(* PLC project Unnamed, Unknown Unnamed 1 *)
(* stored: creationDateTime 2026-06-06T03:01:27, modificationDateTime 2026-06-06T03:01:27 *)

PROGRAM main
  VAR
    conveyor AT %QX0.0 : BOOL;  (* the entry conveyor that transport the boxes to the chain transfer *)
    Load AT %QX0.1 : BOOL;  (* the conveyor on the chain transfer that move the boxes to the right place to be then transported *)
    TransferLeft AT %QX0.3 : BOOL;  (* moves the boxes on the chain transfer to the left *)
    TransferRight AT %QX0.4 : BOOL;  (* moves the boxes on the chain transfer to the right *)
    ConveyoerLeft AT %QX0.5 : BOOL;  (* moves the short boxes to the remover where they get disposed *)
    conveyorRight AT %QX0.6 : BOOL;  (* moves the tall boxes to the remover where they get disposed *)
    HighSensor AT %IX0.0 : BOOL;  (* detects if the boxes are tall *)
    LowSensor AT %IX0.1 : BOOL;  (* detects if the boxes are tall ( the high sensor also need to be false for this to be useful ) *)
    PalletSensor AT %IX0.2 : BOOL;  (* detects the pallet to know to when to start the transportation *)
    Loaded AT %IX0.3 : BOOL;  (* sensor to detect the box is in the right place to be transported *)
    LeftEntry AT %IX0.4 : BOOL;  (* A sensor to to detect that the box has left the chain transfer and reached the left conveyor *)
    at_right_entry AT %IX0.6 : BOOL;  (* A sensor to to detect that the box has left the chain transfer and reached the right conveyor *)
  END_VAR
  VAR
    highsensor_memorybit : BOOL;  (* a boolean variable to save the state of the tall boxes *)
    lowsensor_memorybit : BOOL;  (* a boolean variable to save the state of the short boxes *)
    F_TRIG0 : F_TRIG;
    F_TRIG1 : F_TRIG;
    F_TRIG2 : F_TRIG;
    F_TRIG3 : F_TRIG;
    F_TRIG4 : F_TRIG;
    F_TRIG5 : F_TRIG;
    F_TRIG6 : F_TRIG;
    F_TRIG7 : F_TRIG;
    R_TRIG0 : R_TRIG;
  END_VAR

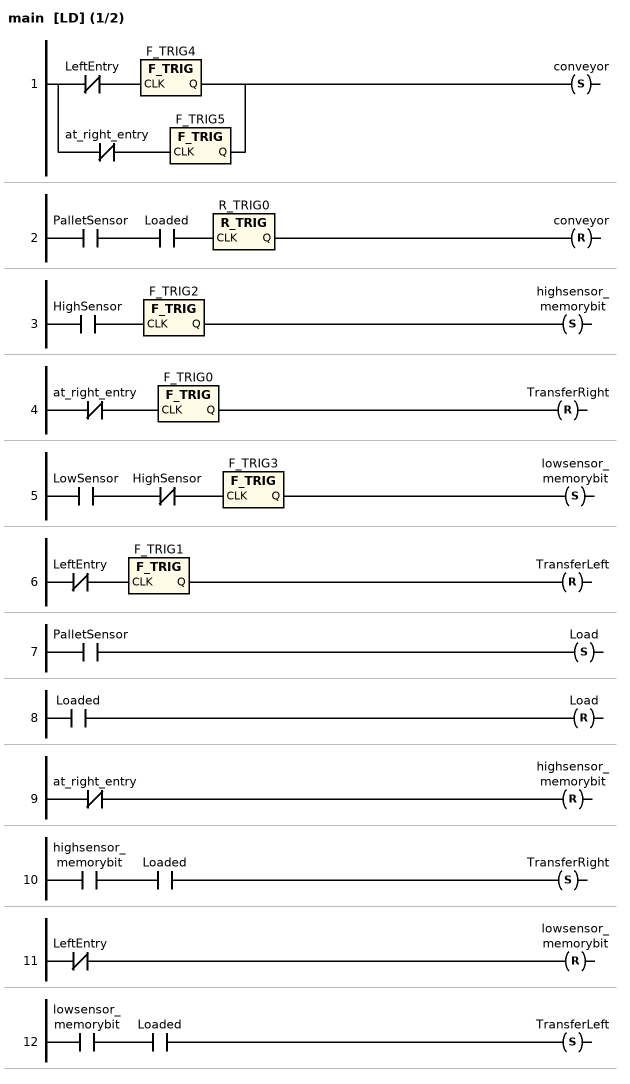
(* LD diagram, written out as Structured Text *)
IF TRUE THEN conveyor := TRUE; END_IF;
IF TRUE THEN ConveyoerLeft := TRUE; END_IF;
IF TRUE THEN conveyorRight := TRUE; END_IF;
F_TRIG4(CLK := NOT LeftEntry);
F_TRIG5(CLK := NOT at_right_entry);
IF F_TRIG4.Q OR F_TRIG5.Q THEN conveyor := TRUE; END_IF;
R_TRIG0(CLK := PalletSensor AND Loaded);
IF R_TRIG0.Q THEN conveyor := FALSE; END_IF;
IF PalletSensor THEN Load := TRUE; END_IF;
IF Loaded THEN Load := FALSE; END_IF;
F_TRIG2(CLK := HighSensor);
IF F_TRIG2.Q THEN highsensor_memorybit := TRUE; END_IF;
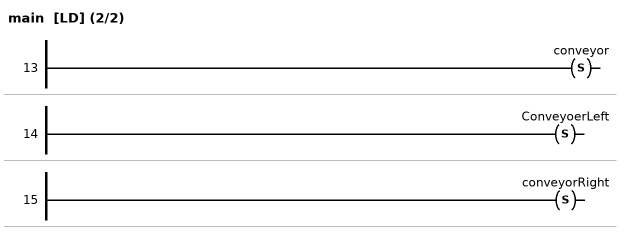
IF NOT at_right_entry THEN highsensor_memorybit := FALSE; END_IF;
IF highsensor_memorybit AND Loaded THEN TransferRight := TRUE; END_IF;
F_TRIG0(CLK := NOT at_right_entry);
IF F_TRIG0.Q THEN TransferRight := FALSE; END_IF;
F_TRIG3(CLK := LowSensor AND NOT HighSensor);
IF F_TRIG3.Q THEN lowsensor_memorybit := TRUE; END_IF;
IF NOT LeftEntry THEN lowsensor_memorybit := FALSE; END_IF;
IF lowsensor_memorybit AND Loaded THEN TransferLeft := TRUE; END_IF;
F_TRIG1(CLK := NOT LeftEntry);
IF F_TRIG1.Q THEN TransferLeft := FALSE; END_IF;
END_PROGRAM

CONFIGURATION Config0
  RESOURCE Res0 ON PLC
    TASK task0(INTERVAL := T#20ms, PRIORITY := 1);
    PROGRAM instance0 WITH task0 : main;
  END_RESOURCE
END_CONFIGURATION
